// TwinCAT 3 PLC project OSCAT
// Title: OSCAT
// Company: RWTH Aachen University - E.ON Energy Research Center
// ProjectVersion: 1.1.3
// Description: This library is based on the OSCAT library (http://www.oscat.de/)
// ProgramVersion: 3.1.4022.1
// libraries:
//   Tc2_Standard, * (Beckhoff Automation GmbH)
// project tree:
//   oscat_basic/Data types/ CALENDAR.TcDUT (not stored), COMPLEX.TcDUT (not stored), CONSTANTS_LANGUAGE.TcDUT (not stored), CONSTANTS_LOCATION.TcDUT (not stored), CONSTANTS_MATH.TcDUT (not stored), CONSTANTS_PHYS.TcDUT (not stored), CONSTANTS_SETUP.TcDUT (not stored), ESR_DATA.TcDUT (not stored), CONTROL_MODE.TcDUT (not stored), FRACTION.TcDUT (not stored), HOLIDAY_DATA.TcDUT (not stored), REAL2.TcDUT (not stored), SDT.TcDUT (not stored), CONTROL_PARAMETERS.TcDUT (not stored), IO_TERMINAL_PARAMETERS.TcDUT (not stored), TIMER_EVENT.TcDUT (not stored), VECTOR_3.TcDUT (not stored)
//   oscat_basic/Global Variables/ Constants_2.TcGVL (not stored), Globale_Variablen_2.TcGVL (not stored)
//   oscat_basic/POUs/Buffer Management/ BUFFER_COMP.TcPOU (not stored), BUFFER_SEARCH.TcPOU (not stored), BUFFER_TO_STRING.TcPOU (not stored), _BUFFER_INSERT.TcPOU (not stored), _BUFFER_UPPERCASE.TcPOU (not stored), _STRING_TO_BUFFER.TcPOU (not stored)
//   oscat_basic/POUs/Engineering/automation/ DRIVER_1.TcPOU (not stored), DRIVER_4.TcPOU (not stored), DRIVER_4C.TcPOU (not stored), FLOW_CONTROL.TcPOU (not stored), FT_Profile.TcPOU (not stored), INC_DEC.TcPOU (not stored), INTERLOCK.TcPOU (not stored), INTERLOCK_4.TcPOU (not stored), MANUAL.TcPOU (not stored), MANUAL_1.TcPOU (not stored), MANUAL_2.TcPOU (not stored), MANUAL_4.TcPOU (not stored), PARSET.TcPOU (not stored), PARSET2.TcPOU (not stored), SIGNAL.TcPOU (not stored), SIGNAL_4.TcPOU (not stored), SRAMP.TcPOU (not stored), TUNE.TcPOU (not stored), TUNE2.TcPOU (not stored)
//   oscat_basic/POUs/Engineering/Control/ BAND_B.TcPOU (not stored), CONTROL_SET1.TcPOU (not stored), CONTROL_SET2.TcPOU (not stored), CTRL_IN.TcPOU (not stored), CTRL_OUT.TcPOU (not stored), CTRL_PI.TcPOU (not stored), CTRL_PID.TcPOU (not stored), CTRL_PWM.TcPOU (not stored), DEAD_BAND.TcPOU (not stored), DEAD_BAND_A.TcPOU (not stored), DEAD_ZONE.TcPOU (not stored), DEAD_ZONE2.TcPOU (not stored), VOLTAGE_CONTROL.TcPOU (not stored), FB_CONTROL.TcPOU (not stored), FB_Integrate.TcPOU (not stored), FB_PID.TcPOU (not stored), FT_DERIV.TcPOU (not stored), FT_IMP.TcPOU (not stored), FT_INT.TcPOU (not stored), FT_INT2.TcPOU (not stored), FT_PD.TcPOU (not stored), FT_PDT1.TcPOU (not stored), FT_PI.TcPOU (not stored), FT_PID.TcPOU (not stored), FT_PIDW.TcPOU (not stored), FT_PIDWL.TcPOU (not stored), FT_PIW.TcPOU (not stored), FT_PIWL.TcPOU (not stored), FT_PT1.TcPOU (not stored), FT_PT2.TcPOU (not stored), FT_TN16.TcPOU (not stored), FT_TN64.TcPOU (not stored), FT_TN8.TcPOU (not stored), HYST.TcPOU (not stored), HYST_1.TcPOU (not stored), HYST_2.TcPOU (not stored), HYST_3.TcPOU (not stored), INTEGRATE.TcPOU (not stored)
//   oscat_basic/POUs/Engineering/Conversion/ ASTRO.TcPOU (not stored), BFT_TO_MS.TcPOU (not stored), C_TO_F.TcPOU (not stored), C_TO_K.TcPOU (not stored), DEG_TO_DIR.TcPOU (not stored), DIR_TO_DEG.TcPOU (not stored), ENERGY.TcPOU (not stored), F_TO_C.TcPOU (not stored), F_TO_OM.TcPOU (not stored), F_TO_PT.TcPOU (not stored), GEO_TO_DEG.TcPOU (not stored), KMH_TO_MS.TcPOU (not stored), K_TO_C.TcPOU (not stored), LENGTH.TcPOU (not stored), MS_TO_BFT.TcPOU (not stored), MS_TO_KMH.TcPOU (not stored), OM_TO_F.TcPOU (not stored), PRESSURE.TcPOU (not stored), PT_TO_F.TcPOU (not stored), SPEED.TcPOU (not stored), TEMPERATURE.TcPOU (not stored)
//   oscat_basic/POUs/Engineering/measurements/ ALARM_2.TcPOU (not stored), BAR_GRAPH.TcPOU (not stored), CALIBRATE.TcPOU (not stored), CYCLE_TIME.TcPOU (not stored), DT_SIMU.TcPOU (not stored), FLOW_METER.TcPOU (not stored), METER.TcPOU (not stored), METER_STAT.TcPOU (not stored), M_D.TcPOU (not stored), M_T.TcPOU (not stored), M_TX.TcPOU (not stored), ONTIME.TcPOU (not stored), TC_MS.TcPOU (not stored), TC_S.TcPOU (not stored), TC_US.TcPOU (not stored), T_PLC_MS.TcPOU (not stored), T_PLC_US.TcPOU (not stored)
//   oscat_basic/POUs/Engineering/sensor/ MULTI_IN.TcPOU (not stored), RES_NI.TcPOU (not stored), RES_NTC.TcPOU (not stored), RES_PT.TcPOU (not stored), RES_SI.TcPOU (not stored), SENSOR_INT.TcPOU (not stored), TEMP_NI.TcPOU (not stored), TEMP_NTC.TcPOU (not stored), TEMP_PT.TcPOU (not stored), TEMP_SI.TcPOU (not stored)
//   oscat_basic/POUs/Engineering/signal generators/ GEN_PULSE.TcPOU (not stored), GEN_PW2.TcPOU (not stored), GEN_RDM.TcPOU (not stored), GEN_RDT.TcPOU (not stored), GEN_RMP.TcPOU (not stored), GEN_SIN.TcPOU (not stored), GEN_SQR.TcPOU (not stored), PWM_DC.TcPOU (not stored), PWM_PW.TcPOU (not stored), RMP_B.TcPOU (not stored), RMP_SOFT.TcPOU (not stored), RMP_W.TcPOU (not stored), _RMP_B.TcPOU (not stored), _RMP_NEXT.TcPOU (not stored), _RMP_W.TcPOU (not stored)
//   oscat_basic/POUs/Engineering/signal processing/ AIN.TcPOU (not stored), AIN1.TcPOU (not stored), AOUT.TcPOU (not stored), AOUT1.TcPOU (not stored), BYTE_TO_RANGE.TcPOU (not stored), DELAY.TcPOU (not stored), DELAY_200.TcPOU (not stored), DELAY_4.TcPOU (not stored), FADE.TcPOU (not stored), FB_InLinear.TcPOU (not stored), FB_InOnOff.TcPOU (not stored), FB_OutLinear.TcPOU (not stored), FB_OutOnOff.TcPOU (not stored), FILTER_DW.TcPOU (not stored), FILTER_I.TcPOU (not stored), FILTER_MAV_DW.TcPOU, FILTER_MAV_W.TcPOU (not stored), FILTER_W.TcPOU (not stored), FILTER_WAV.TcPOU (not stored), MIX.TcPOU (not stored), MUX_R2.TcPOU (not stored), MUX_R4.TcPOU (not stored), OFFSET.TcPOU (not stored), OFFSET2.TcPOU (not stored), OVERRIDE.TcPOU (not stored), RANGE_TO_BYTE.TcPOU (not stored), RANGE_TO_WORD.TcPOU (not stored), SCALE.TcPOU (not stored), SCALE_B.TcPOU (not stored), SCALE_B2.TcPOU (not stored), SCALE_B4.TcPOU (not stored), SCALE_B8.TcPOU (not stored), SCALE_D.TcPOU (not stored), SCALE_R.TcPOU (not stored), SCALE_X2.TcPOU (not stored), SCALE_X4.TcPOU (not stored), SCALE_X8.TcPOU (not stored), SEL2_OF_3.TcPOU (not stored), SEL2_OF_3B.TcPOU (not stored), SH.TcPOU (not stored), SH_1.TcPOU (not stored), SH_2.TcPOU (not stored), SH_T.TcPOU (not stored), STAIR.TcPOU (not stored), STAIR2.TcPOU (not stored), TREND.TcPOU (not stored), TREND_DW.TcPOU (not stored), WORD_TO_RANGE.TcPOU (not stored)
//   oscat_basic/POUs/List Processing/ LIST_ADD.TcPOU (not stored), LIST_CLEAN.TcPOU (not stored), LIST_GET.TcPOU (not stored), LIST_INSERT.TcPOU (not stored), LIST_LEN.TcPOU (not stored), LIST_NEXT.TcPOU (not stored), LIST_RETRIEVE.TcPOU (not stored), LIST_RETRIEVE_LAST.TcPOU (not stored)
//   oscat_basic/POUs/Logic/FF edge triggered/ COUNT_BR.TcPOU (not stored), COUNT_DR.TcPOU (not stored), FF_D2E.TcPOU (not stored), FF_D4E.TcPOU (not stored), FF_DRE.TcPOU (not stored), FF_JKE.TcPOU (not stored), FF_RSE.TcPOU (not stored), SELECT_8.TcPOU (not stored), SHR_4E.TcPOU (not stored), SHR_4UDE.TcPOU (not stored), SHR_8PLE.TcPOU (not stored), SHR_8UDE.TcPOU (not stored), TOGGLE.TcPOU (not stored)
//   oscat_basic/POUs/Logic/FF pulse triggered/ LTCH.TcPOU (not stored), LTCH_4.TcPOU (not stored), STORE_8.TcPOU (not stored)
//   oscat_basic/POUs/Logic/gate logic/ BCDC_TO_INT.TcPOU (not stored), BIT_COUNT.TcPOU (not stored), BIT_LOAD_B.TcPOU (not stored), BIT_LOAD_B2.TcPOU (not stored), BIT_LOAD_DW.TcPOU (not stored), BIT_LOAD_DW2.TcPOU (not stored), BIT_LOAD_W.TcPOU (not stored), BIT_LOAD_W2.TcPOU (not stored), BIT_OF_DWORD.TcPOU (not stored), BIT_TOGGLE_B.TcPOU (not stored), BIT_TOGGLE_DW.TcPOU (not stored), BIT_TOGGLE_W.TcPOU (not stored), BYTE_OF_BIT.TcPOU (not stored), BYTE_OF_DWORD.TcPOU (not stored), BYTE_TO_BITS.TcPOU (not stored), BYTE_TO_GRAY.TcPOU (not stored), CHECK_PARITY.TcPOU (not stored), CHK_REAL.TcPOU (not stored), DEC_2.TcPOU (not stored), DEC_4.TcPOU (not stored), DEC_8.TcPOU (not stored), DWORD_OF_BYTE.TcPOU (not stored), DWORD_OF_WORD.TcPOU (not stored), DW_TO_REAL.TcPOU (not stored), GRAY_TO_BYTE.TcPOU (not stored), INT_TO_BCDC.TcPOU (not stored), MUX_2.TcPOU (not stored), MUX_4.TcPOU (not stored), PARITY.TcPOU (not stored), REAL_TO_DW.TcPOU (not stored), REFLECT.TcPOU (not stored), REVERSE.TcPOU (not stored), SHL1.TcPOU (not stored), SHR1.TcPOU (not stored), SWAP_BYTE.TcPOU (not stored), SWAP_BYTE2.TcPOU (not stored), WORD_OF_BYTE.TcPOU (not stored), WORD_OF_DWORD.TcPOU (not stored)
//   oscat_basic/POUs/Logic/generators/ A_TRIG.TcPOU (not stored), B_TRIG.TcPOU (not stored), CLICK_CNT.TcPOU (not stored), CLICK_DEC.TcPOU (not stored), CLK_DIV.TcPOU (not stored), CLK_N.TcPOU (not stored), CLK_PRG.TcPOU (not stored), CLK_PULSE.TcPOU (not stored), CYCLE_4.TcPOU (not stored), D_TRIG.TcPOU (not stored), GEN_BIT.TcPOU (not stored), GEN_SQ.TcPOU (not stored), SCHEDULER.TcPOU (not stored), SCHEDULER_2.TcPOU (not stored), SEQUENCE_4.TcPOU (not stored), SEQUENCE_64.TcPOU (not stored), SEQUENCE_8.TcPOU (not stored), TMAX.TcPOU (not stored), TMIN.TcPOU (not stored), TOF_1.TcPOU (not stored), TONOF.TcPOU (not stored), TP_1.TcPOU (not stored), TP_1D.TcPOU (not stored), TP_X.TcPOU (not stored)
//   oscat_basic/POUs/Logic/memory/ FIFO_16.TcPOU (not stored), FIFO_32.TcPOU (not stored), STACK_16.TcPOU (not stored), STACK_32.TcPOU (not stored)
//   oscat_basic/POUs/Logic/Others/ CRC_GEN.TcPOU (not stored), MATRIX.TcPOU (not stored), PIN_CODE.TcPOU (not stored)
//   oscat_basic/POUs/Mathematical/ ACOSH.TcPOU (not stored), ACOTH.TcPOU (not stored), AGDF.TcPOU (not stored), ASINH.TcPOU (not stored), ATAN2.TcPOU (not stored), ATANH.TcPOU (not stored), BETA.TcPOU (not stored), BINOM.TcPOU (not stored), CAUCHY.TcPOU (not stored), CAUCHYCD.TcPOU (not stored), CEIL.TcPOU (not stored), CEIL2.TcPOU (not stored), CMP.TcPOU (not stored), COSH.TcPOU (not stored), COTH.TcPOU (not stored), DEC1.TcPOU (not stored), DEG.TcPOU (not stored), DIFFER.TcPOU (not stored), D_TRUNC.TcPOU (not stored), ERF.TcPOU (not stored), ERFC.TcPOU (not stored), EVEN.TcPOU (not stored), EXP10.TcPOU (not stored), EXPN.TcPOU (not stored), FACT.TcPOU (not stored), FIB.TcPOU (not stored), FLOOR.TcPOU (not stored), FLOOR2.TcPOU (not stored), FRACT.TcPOU (not stored), GAMMA.TcPOU (not stored), GAUSS.TcPOU (not stored), GAUSSCD.TcPOU (not stored), GCD.TcPOU (not stored), GDF.TcPOU (not stored), GOLD.TcPOU (not stored), HYPOT.TcPOU (not stored), INC.TcPOU (not stored), INC1.TcPOU (not stored), INC2.TcPOU (not stored), INV.TcPOU (not stored), LAMBERT_W.TcPOU (not stored), LANGEVIN.TcPOU (not stored), MAX3.TcPOU (not stored), MID3.TcPOU (not stored), MIN3.TcPOU (not stored), MODR.TcPOU (not stored), MUL_ADD.TcPOU (not stored), NEGX.TcPOU (not stored), RAD.TcPOU (not stored), RDM.TcPOU (not stored), RDM2.TcPOU (not stored), RDMDW.TcPOU (not stored), REAL_TO_FRAC.TcPOU (not stored), RND.TcPOU (not stored), ROUND.TcPOU (not stored), SGN.TcPOU (not stored), SIGMOID.TcPOU (not stored), SIGN_I.TcPOU (not stored), SIGN_R.TcPOU (not stored), SINC.TcPOU (not stored), SINH.TcPOU (not stored), SQRTN.TcPOU (not stored), TANC.TcPOU (not stored), TANH.TcPOU (not stored), WINDOW.TcPOU (not stored), WINDOW2.TcPOU (not stored)
//   oscat_basic/POUs/Mathematical/Array/ ARRAY_AVG.TcPOU (not stored), ARRAY_GAV.TcPOU (not stored), ARRAY_HAV.TcPOU (not stored), ARRAY_MAX.TcPOU (not stored), ARRAY_MIN.TcPOU (not stored), ARRAY_SDV.TcPOU (not stored), ARRAY_SPR.TcPOU (not stored), ARRAY_SUM.TcPOU (not stored), ARRAY_TREND.TcPOU (not stored), ARRAY_VAR.TcPOU (not stored), IS_SORTED.TcPOU (not stored), _ARRAY_ABS.TcPOU (not stored), _ARRAY_ADD.TcPOU (not stored), _ARRAY_INIT.TcPOU (not stored), _ARRAY_MEDIAN.TcPOU (not stored), _ARRAY_MUL.TcPOU (not stored), _ARRAY_SHUFFLE.TcPOU (not stored), _ARRAY_SORT.TcPOU (not stored)
//   oscat_basic/POUs/Mathematical/Complex/ CABS.TcPOU (not stored), CACOS.TcPOU (not stored), CACOSH.TcPOU (not stored), CADD.TcPOU (not stored), CARG.TcPOU (not stored), CASIN.TcPOU (not stored), CASINH.TcPOU (not stored), CATAN.TcPOU (not stored), CATANH.TcPOU (not stored), CCON.TcPOU (not stored), CCOS.TcPOU (not stored), CCOSH.TcPOU (not stored), CDIV.TcPOU (not stored), CEXP.TcPOU (not stored), CINV.TcPOU (not stored), CLOG.TcPOU (not stored), CMUL.TcPOU (not stored), CPOL.TcPOU (not stored), CPOW.TcPOU (not stored), CSET.TcPOU (not stored), CSIN.TcPOU (not stored), CSINH.TcPOU (not stored), CSQRT.TcPOU (not stored), CSUB.TcPOU (not stored), CTAN.TcPOU (not stored), CTANH.TcPOU (not stored)
//   oscat_basic/POUs/Mathematical/Double Precision/ R2_ABS.TcPOU (not stored), R2_ADD.TcPOU (not stored), R2_ADD2.TcPOU (not stored), R2_MUL.TcPOU (not stored), R2_SET.TcPOU (not stored)
//   oscat_basic/POUs/Mathematical/functions/ FRMP_B.TcPOU (not stored), FT_AVG.TcPOU (not stored), FT_AVG_200.TcPOU (not stored), FT_MIN_MAX.TcPOU (not stored), FT_RMP.TcPOU (not stored), F_LIN.TcPOU (not stored), F_LIN2.TcPOU (not stored), F_POLY.TcPOU (not stored), F_POWER.TcPOU (not stored), F_QUAD.TcPOU (not stored), LINEAR_INT.TcPOU (not stored), POLYNOM_INT.TcPOU (not stored)
//   oscat_basic/POUs/Mathematical/Geometry/ CIRCLE_A.TcPOU (not stored), CIRCLE_C.TcPOU (not stored), CIRCLE_SEG.TcPOU (not stored), CONE_V.TcPOU (not stored), ELLIPSE_A.TcPOU (not stored), ELLIPSE_C.TcPOU (not stored), SPHERE_V.TcPOU (not stored), TRIANGLE_A.TcPOU (not stored)
//   oscat_basic/POUs/Mathematical/Vektormathematik/ V3_ABS.TcPOU (not stored), V3_ADD.TcPOU (not stored), V3_ANG.TcPOU (not stored), V3_DPRO.TcPOU (not stored), V3_NORM.TcPOU (not stored), V3_NUL.TcPOU (not stored), V3_PAR.TcPOU (not stored), V3_REV.TcPOU (not stored), V3_SMUL.TcPOU (not stored), V3_SUB.TcPOU (not stored), V3_XANG.TcPOU (not stored), V3_XPRO.TcPOU (not stored), V3_YANG.TcPOU (not stored), V3_ZANG.TcPOU (not stored)
//   oscat_basic/POUs/Other/ ESR_COLLECT.TcPOU (not stored), ESR_MON_B8.TcPOU (not stored), ESR_MON_R4.TcPOU (not stored), ESR_MON_X8.TcPOU (not stored), OSCAT_VERSION.TcPOU (not stored), STATUS_TO_ESR.TcPOU (not stored)
//   oscat_basic/POUs/String/ BIN_TO_BYTE.TcPOU (not stored), BIN_TO_DWORD.TcPOU (not stored), BYTE_TO_STRB.TcPOU (not stored), BYTE_TO_STRH.TcPOU (not stored), CAPITALIZE.TcPOU (not stored), CHARCODE.TcPOU (not stored), CHARNAME.TcPOU (not stored), CHR_TO_STRING.TcPOU (not stored), CLEAN.TcPOU (not stored), CODE.TcPOU (not stored), COUNT_CHAR.TcPOU (not stored), COUNT_SUBSTRING.TcPOU (not stored), DEC_TO_BYTE.TcPOU (not stored), DEC_TO_DWORD.TcPOU (not stored), DEC_TO_INT.TcPOU (not stored), DEL_CHARS.TcPOU (not stored), DT_TO_STRF.TcPOU (not stored), DWORD_TO_STRB.TcPOU (not stored), DWORD_TO_STRF.TcPOU (not stored), DWORD_TO_STRH.TcPOU (not stored), EXEC.TcPOU (not stored), FILL.TcPOU (not stored), FINDB.TcPOU (not stored), FINDB_NONUM.TcPOU (not stored), FINDB_NUM.TcPOU (not stored), FINDP.TcPOU (not stored), FIND_CHAR.TcPOU (not stored), FIND_CTRL.TcPOU (not stored), FIND_NONUM.TcPOU (not stored), FIND_NUM.TcPOU (not stored), FIX.TcPOU (not stored), FLOAT_TO_REAL.TcPOU (not stored), FSTRING_TO_BYTE.TcPOU (not stored), FSTRING_TO_DT.TcPOU (not stored), FSTRING_TO_DWORD.TcPOU (not stored), FSTRING_TO_MONTH.TcPOU (not stored), FSTRING_TO_WEEK.TcPOU (not stored), FSTRING_TO_WEEKDAY.TcPOU (not stored), HEX_TO_BYTE.TcPOU (not stored), HEX_TO_DWORD.TcPOU (not stored), ISC_ALPHA.TcPOU (not stored), ISC_CTRL.TcPOU (not stored), ISC_HEX.TcPOU (not stored), ISC_LOWER.TcPOU (not stored), ISC_NUM.TcPOU (not stored), ISC_UPPER.TcPOU (not stored), IS_ALNUM.TcPOU (not stored), IS_ALPHA.TcPOU (not stored), IS_CC.TcPOU (not stored), IS_CTRL.TcPOU (not stored), IS_HEX.TcPOU (not stored), IS_LOWER.TcPOU (not stored), IS_NCC.TcPOU (not stored), IS_NUM.TcPOU (not stored), IS_UPPER.TcPOU (not stored), LOWERCASE.TcPOU (not stored), MESSAGE_4R.TcPOU (not stored), MESSAGE_8.TcPOU (not stored), MIRROR.TcPOU (not stored), MONTH_TO_STRING.TcPOU (not stored), OCT_TO_BYTE.TcPOU (not stored), OCT_TO_DWORD.TcPOU (not stored), REAL_TO_STRF.TcPOU (not stored), REPLACE_ALL.TcPOU (not stored), REPLACE_CHARS.TcPOU (not stored), REPLACE_UML.TcPOU (not stored), TICKER.TcPOU (not stored), TO_LOWER.TcPOU (not stored), TO_UML.TcPOU (not stored), TO_UPPER.TcPOU (not stored), TRIM.TcPOU (not stored), TRIM1.TcPOU (not stored), TRIME.TcPOU (not stored), UPPERCASE.TcPOU (not stored), WEEKDAY_TO_STRING.TcPOU (not stored)
//   oscat_basic/POUs/Time&Date/ CALENDAR_CALC.TcPOU (not stored), DATE_ADD.TcPOU (not stored), DAYS_DELTA.TcPOU (not stored), DAYS_IN_MONTH.TcPOU (not stored), DAYS_IN_YEAR.TcPOU (not stored), DAY_OF_DATE.TcPOU (not stored), DAY_OF_MONTH.TcPOU (not stored), DAY_OF_WEEK.TcPOU (not stored), DAY_OF_YEAR.TcPOU (not stored), DAY_TO_TIME.TcPOU (not stored), DCF77.TcPOU (not stored), DST.TcPOU (not stored), DT2_TO_SDT.TcPOU (not stored), DT_TO_SDT.TcPOU (not stored), EASTER.TcPOU (not stored), EVENTS.TcPOU (not stored), HOLIDAY.TcPOU (not stored), HOUR.TcPOU (not stored), HOUR_OF_DT.TcPOU (not stored), HOUR_TO_TIME.TcPOU (not stored), HOUR_TO_TOD.TcPOU (not stored), JD2000.TcPOU (not stored), LEAP_DAY.TcPOU (not stored), LEAP_OF_DATE.TcPOU (not stored), LEAP_YEAR.TcPOU (not stored), LTIME_TO_UTC.TcPOU (not stored), MINUTE.TcPOU (not stored), MINUTE_OF_DT.TcPOU (not stored), MINUTE_TO_TIME.TcPOU (not stored), MONTH_BEGIN.TcPOU (not stored), MONTH_END.TcPOU (not stored), MONTH_OF_DATE.TcPOU (not stored), MULTIME.TcPOU (not stored), PERIOD.TcPOU (not stored), PERIOD2.TcPOU (not stored), REFRACTION.TcPOU (not stored), RTC_2.TcPOU (not stored), RTC_MS.TcPOU (not stored), SDT_TO_DATE.TcPOU (not stored), SDT_TO_DT.TcPOU (not stored), SDT_TO_TOD.TcPOU (not stored), SECOND.TcPOU (not stored), SECOND_OF_DT.TcPOU (not stored), SECOND_TO_TIME.TcPOU (not stored), SET_DATE.TcPOU (not stored), SET_DT.TcPOU (not stored), SET_TOD.TcPOU (not stored), SUN_MIDDAY.TcPOU (not stored), SUN_POS.TcPOU (not stored), SUN_TIME.TcPOU (not stored), TIMECHECK.TcPOU (not stored), TON_P.TcPOU (not stored), UTC_TO_LTIME.TcPOU (not stored), WORK_WEEK.TcPOU (not stored), YEAR_BEGIN.TcPOU (not stored), YEAR_END.TcPOU (not stored), YEAR_OF_DATE.TcPOU (not stored)
//   oscat_building/Global Variables/ Constants.TcGVL (not stored), Globale_Variablen.TcGVL (not stored), Setup_Data.TcGVL (not stored)
//   oscat_building/POUs/actuators/ ACTUATOR_2P.TcPOU (not stored), ACTUATOR_3P.TcPOU (not stored), ACTUATOR_A.TcPOU (not stored), ACTUATOR_COIL.TcPOU (not stored), ACTUATOR_PUMP.TcPOU (not stored), ACTUATOR_UD.TcPOU (not stored), AUTORUN.TcPOU (not stored)
//   oscat_building/POUs/electrical/ CLICK.TcPOU (not stored), CLICK_MODE.TcPOU (not stored), DEBOUNCE.TcPOU (not stored), DIMM_2.TcPOU (not stored), DIMM_I.TcPOU (not stored), F_LAMP.TcPOU (not stored), PULSE_LENGTH.TcPOU (not stored), PULSE_T.TcPOU (not stored), SWITCH_I.TcPOU (not stored), SWITCH_X.TcPOU (not stored), SW_RECONFIG.TcPOU (not stored), TIMER_1.TcPOU (not stored), TIMER_2.TcPOU (not stored), TIMER_EVENT_DECODE.TcPOU (not stored), TIMER_EXT.TcPOU (not stored), TIMER_P4.TcPOU (not stored)
//   oscat_building/POUs/HLK/ AIR_DENSITY.TcPOU (not stored), AIR_ENTHALPY.TcPOU (not stored), BOILER.TcPOU (not stored), BURNER.TcPOU (not stored), DEW_CON.TcPOU (not stored), DEW_RH.TcPOU (not stored), DEW_TEMP.TcPOU (not stored), HEAT_INDEX.TcPOU (not stored), HEAT_METER.TcPOU (not stored), HEAT_TEMP.TcPOU (not stored), LEGIONELLA.TcPOU (not stored), SDD.TcPOU (not stored), SDD_NH3.TcPOU (not stored), SDT_NH3.TcPOU (not stored), TANK_LEVEL.TcPOU (not stored), TANK_VOL1.TcPOU (not stored), TANK_VOL2.TcPOU (not stored), TEMP_EXT.TcPOU (not stored), T_AVG24.TcPOU (not stored), WATER_CP.TcPOU (not stored), WATER_DENSITY.TcPOU (not stored), WATER_ENTHALPY.TcPOU (not stored), WCT.TcPOU (not stored)
//   oscat_building/POUs/Jalousie/ BLIND_ACTUATOR.TcPOU (not stored), BLIND_CONTROL.TcPOU (not stored), BLIND_CONTROL_S.TcPOU (not stored), BLIND_INPUT.TcPOU (not stored), BLIND_NIGHT.TcPOU (not stored), BLIND_SCENE.TcPOU (not stored), BLIND_SECURITY.TcPOU (not stored), BLIND_SET.TcPOU (not stored), BLIND_SHADE.TcPOU (not stored), BLIND_SHADE_S.TcPOU (not stored)
//   oscat_building/POUs/Other/ BUILDING_VERSION.TcPOU (not stored)
//   oscat_network/Data types/DATA_LOG/ DLOG_DATA.TcDUT (not stored), LOG_CONTROL.TcDUT (not stored), MYSQL_COM.TcDUT (not stored), PRINTF_DATA.TcDUT (not stored), UNI_CIRCULAR_BUFFER_DATA.TcDUT (not stored), us_LOG_VIEWPORT.TcDUT (not stored)
//   oscat_network/Data types/FILE_SERVER/ FILE_PATH_DATA.TcDUT (not stored), FILE_SERVER_DATA.TcDUT (not stored)
//   oscat_network/Data types/NETWORK/ IP2GEO_DATA.TcDUT (not stored), IP_C.TcDUT (not stored), IP_FIFO_DATA.TcDUT (not stored), NETWORK_BUFFER.TcDUT (not stored), NETWORK_BUFFER_SHORT.TcDUT (not stored), NW_BUF_LONG.TcDUT (not stored), NW_BUF_SHORT.TcDUT (not stored), URL.TcDUT (not stored), VMAP_DATA.TcDUT (not stored), XML_CONTROL.TcDUT (not stored)
//   oscat_network/Data types/NET_VAR/ NET_VAR_DATA.TcDUT (not stored)
//   oscat_network/Data types/TELNET_VISION/ us_TN_INPUT_CONTROL.TcDUT (not stored), us_TN_INPUT_CONTROL_DATA.TcDUT (not stored), us_TN_MENU.TcDUT (not stored), us_TN_MENU_POPUP.TcDUT (not stored), us_TN_SCREEN.TcDUT (not stored)
//   oscat_network/Data types/WEATHER/ WORLD_WEATHER_CUR.TcDUT (not stored), WORLD_WEATHER_DATA.TcDUT (not stored), WORLD_WEATHER_DAY.TcDUT (not stored), YAHOO_WEATHER_DATA.TcDUT (not stored)
//   oscat_network/Global Variables/ Constants_1.TcGVL (not stored), Globale_Variablen_1.TcGVL (not stored)
//   oscat_network/POUs/CO_NVERT/ BASE64_DECODE_STREAM_1.TcPOU (not stored), BASE64_DECODE_STR_1.TcPOU (not stored), BASE64_ENCODE_STREAM_1.TcPOU (not stored), BASE64_ENCODE_STR_1.TcPOU (not stored), HTML_DECODE_1.TcPOU (not stored), HTML_ENCODE_1.TcPOU (not stored), IP4_CHECK_1.TcPOU (not stored), IP4_DECODE_1.TcPOU (not stored), IP4_TO_STRING_1.TcPOU (not stored), IS_IP4_1.TcPOU (not stored), IS_URLCHR_1.TcPOU (not stored), MD5_AUX_1.TcPOU (not stored), MD5_CRAM_AUTH_1.TcPOU (not stored), MD5_STREAM_1.TcPOU (not stored), MD5_STR_1.TcPOU (not stored), MD5_TO_STRH_1.TcPOU (not stored), RC4_CRYPT_STREAM_1.TcPOU (not stored), SHA1_STREAM_1.TcPOU (not stored), SHA1_STR_1.TcPOU (not stored), SHA1_TO_STRH_1.TcPOU (not stored), STRING_TO_URL_1.TcPOU (not stored), URL_DECODE_1.TcPOU (not stored), URL_ENCODE_1.TcPOU (not stored), URL_TO_STRING_1.TcPOU (not stored)
//   oscat_network/POUs/DATA_LOG/ DLOG_BOOL_1.TcPOU (not stored), DLOG_DINT_1.TcPOU (not stored), DLOG_DT_1.TcPOU (not stored), DLOG_FILE_TO_FTP_1.TcPOU (not stored), DLOG_FILE_TO_SMTP_1.TcPOU (not stored), DLOG_REAL_1.TcPOU (not stored), DLOG_STORE_FILE_CSV_1.TcPOU (not stored), DLOG_STORE_FILE_HTML_1.TcPOU (not stored), DLOG_STORE_FILE_XML_1.TcPOU (not stored), DLOG_STORE_RRD_1.TcPOU (not stored), DLOG_STRING_1.TcPOU (not stored), UNI_CIRCULAR_BUFFER_1.TcPOU (not stored)
//   oscat_network/POUs/DEMO/ BASE64_DEMO_1.TcPOU (not stored), CSV_PARSER_BUF_DEMO_1.TcPOU (not stored), CSV_PARSER_FILE_DEMO_1.TcPOU (not stored), DLOG_FILE_CSV_DEMO_1.TcPOU (not stored), DLOG_FILE_CSV_FTP_DEMO_1.TcPOU (not stored), DLOG_FILE_CSV_SMTP_DEMO_1.TcPOU (not stored), DLOG_FILE_HTML_DEMO_1.TcPOU (not stored), DLOG_FILE_XML_DEMO_1.TcPOU (not stored), DLOG_RRD_DEMO_1.TcPOU (not stored), DNS_DYN_DEMO_1.TcPOU (not stored), DNS_REV_DEMO_1.TcPOU (not stored), DNS_SNTP_SYSLOG_DEMO_1.TcPOU (not stored), FILE_BLOCK_DEMO_1.TcPOU (not stored), FTP_CLIENT_DEMO_1.TcPOU (not stored), GET_WAN_IP_DEMO_1.TcPOU (not stored), HTTP_DEMO_1.TcPOU (not stored), INI_PARSER_BUF_DEMO_1.TcPOU (not stored), INI_PARSER_FILE_DEMO_1.TcPOU (not stored), IP2GEO_DEMO_1.TcPOU (not stored), IRTRANS_DEMO_1.TcPOU (not stored), MB_CLIENT_DEMO_1.TcPOU (not stored), MB_SERVER_DEMO_1.TcPOU (not stored), MD5_CRAM_AUTH_DEMO_1.TcPOU (not stored), NET_VAR_MASTER_DEMO_1.TcPOU (not stored), NET_VAR_SLAVE_DEMO_1.TcPOU (not stored), RC4_CRYPT_DEMO_1.TcPOU (not stored), SHA1_MD5_DEMO_1.TcPOU (not stored), SMTP_CLIENT_DEMO_1.TcPOU (not stored), SPIDER_DEMO_1.TcPOU (not stored), TELNET_LOG_DEMO_1.TcPOU (not stored), TELNET_PRINT_DEMO_1.TcPOU (not stored), TN_VISION_DEMO_1_1.TcPOU (not stored), TN_VISION_DEMO_2_1.TcPOU (not stored), WORLD_WEATHER_DEMO_1.TcPOU (not stored), YAHOO_WEATHER_DEMO_1.TcPOU (not stored)
//   oscat_network/POUs/DRIVER/ IRTRANS_DECODE_1.TcPOU (not stored), IRTRANS_RCV_1_1.TcPOU (not stored), IRTRANS_RCV_4_1.TcPOU (not stored), IRTRANS_RCV_8_1.TcPOU (not stored), IRTRANS_SERVER_1.TcPOU (not stored), IRTRANS_SND_1_1.TcPOU (not stored), IRTRANS_SND_4_1.TcPOU (not stored), IRTRANS_SND_8_1.TcPOU (not stored)
//   oscat_network/POUs/FILE/ CSV_PARSER_BUF_1.TcPOU (not stored), CSV_PARSER_FILE_1.TcPOU (not stored), FILE_BLOCK_1.TcPOU (not stored), FILE_PATH_SPLIT_1.TcPOU (not stored), INI_PARSER_BUF_1.TcPOU (not stored), INI_PARSER_FILE_1.TcPOU (not stored)
//   oscat_network/POUs/HARDWARE/ FILE_SERVER_1.TcPOU (not stored), IP_CONTROL2_1.TcPOU (not stored), IP_CONTROL_1.TcPOU (not stored), IP_CONTROL_RESET_1.TcPOU (not stored)
//   oscat_network/POUs/NETWORK/ DNS_CLIENT.TcPOU (not stored), DNS_DYN.TcPOU (not stored), DNS_REV_CLIENT.TcPOU (not stored), FTP_CLIENT.TcPOU (not stored), GET_WAN_IP.TcPOU (not stored), HTTP_GET.TcPOU (not stored), IP2GEO.TcPOU (not stored), IP_FIFO.TcPOU (not stored), LOG_MSG.TcPOU (not stored), LOG_VIEWPORT.TcPOU (not stored), MB_CLIENT.TcPOU (not stored), MB_SERVER.TcPOU (not stored), MB_VMAP.TcPOU (not stored), PRINT_SF.TcPOU (not stored), READ_HTTP.TcPOU (not stored), SMTP_CLIENT.TcPOU (not stored), SNTP_CLIENT.TcPOU (not stored), SNTP_SERVER.TcPOU (not stored), SPIDER_ACCESS.TcPOU (not stored), SYS_LOG.TcPOU (not stored), TELNET_LOG.TcPOU (not stored), TELNET_PRINT.TcPOU (not stored), XML_READER.TcPOU (not stored)
//   oscat_network/POUs/NET_VAR/ NET_VAR_BOOL8.TcPOU (not stored), NET_VAR_BUFFER.TcPOU (not stored), NET_VAR_CONTROL.TcPOU (not stored), NET_VAR_DWORD8.TcPOU (not stored), NET_VAR_REAL8.TcPOU (not stored), NET_VAR_STRING.TcPOU (not stored), NET_VAR_X8.TcPOU (not stored)
//   oscat_network/POUs/OTHER/ ELEMENT_COUNT.TcPOU (not stored), ELEMENT_GET.TcPOU (not stored), NETWORK_VERSION.TcPOU (not stored)
//   oscat_network/POUs/TELNET_VISION/ TN_FRAMEWORK.TcPOU (not stored), TN_INPUT_CONTROL.TcPOU (not stored), TN_INPUT_EDIT_LINE.TcPOU (not stored), TN_INPUT_MENU_BAR.TcPOU (not stored), TN_INPUT_MENU_POPUP.TcPOU (not stored), TN_INPUT_SELECT_POPUP.TcPOU (not stored), TN_INPUT_SELECT_TEXT.TcPOU (not stored), TN_RECEIVE.TcPOU (not stored), TN_SC_ADD_SHADOW.TcPOU (not stored), TN_SC_AREA_RESTORE.TcPOU (not stored), TN_SC_AREA_SAVE.TcPOU (not stored), TN_SC_BOX.TcPOU (not stored), TN_SC_FILL.TcPOU (not stored), TN_SC_LINE.TcPOU (not stored), TN_SC_READ_ATTR.TcPOU (not stored), TN_SC_READ_CHAR.TcPOU (not stored), TN_SC_SHADOW_ATTR.TcPOU (not stored), TN_SC_VIEWPORT.TcPOU (not stored), TN_SC_WRITE.TcPOU (not stored), TN_SC_WRITE_ATTR.TcPOU (not stored), TN_SC_WRITE_C.TcPOU (not stored), TN_SC_WRITE_CHAR.TcPOU (not stored), TN_SC_WRITE_EOS.TcPOU (not stored), TN_SC_XY2_ERROR.TcPOU (not stored), TN_SC_XY_ERROR.TcPOU (not stored), TN_SEND_ROWS.TcPOU (not stored)
//   oscat_network/POUs/WEATHER/ MOON_PHASE.TcPOU (not stored), WORLD_WEATHER.TcPOU (not stored), WORLD_WEATHER_DESC_GE.TcPOU (not stored), WORLD_WEATHER_ICON_OSCAT.TcPOU (not stored), YAHOO_WEATHER.TcPOU (not stored), YAHOO_WEATHER_DESC_GE.TcPOU (not stored), YAHOO_WEATHER_ICON_OSCAT.TcPOU (not stored)

// ---- oscat_basic/POUs/Engineering/signal processing/FILTER_MAV_DW.TcPOU
FUNCTION_BLOCK FILTER_MAV_DW
VAR_INPUT
	X : DWORD;
	N : UINT;
	RST : BOOL;
END_VAR
VAR_OUTPUT
	Y : DWORD;
END_VAR
VAR
	init : BOOL;
	buffer : ARRAY[0..31] OF DWORD;
	i : INT;
	sum : LWORD; 
END_VAR
VAR
	tmp: INT;
END_VAR

(*
version 1.3	23. feb. 2009
programmer 	hugo
tested by		oscat

FILTER_MAV_DW is a moving average filter with programmable length N for DWORD Data.
 
*)

(* limit N to size of buffer *)
N := MIN(N, 32);

(* startup initialisation *)
IF NOT init OR rst OR N = 0 THEN
	init := TRUE;
	tmp := UINT_TO_INT(N)-1;
	FOR i := 0 TO tmp DO
		buffer[i] := X;
	END_FOR;
	sum := Y * N;
	Y := X;
ELSE
	tmp := UINT_TO_INT(N);
	i := INC1(i, tmp);
	sum := sum + X - buffer[i];
	Y := LWORD_TO_DWORD(sum / N);
	buffer[i] := X;
END_IF;




(*
hm 13. oct. 2008	rev 1.0
	original version

hm	27. oct. 2008	rev 1.1
	added typecast to avoid warnings

hm	24. nov. 2008	rev 1.2
	added typecasts to avoid warnings
	avoid divide by 0 if N = 0

hm	23. feb. 2009	rev 1.3
	limit N to max array size

*)

END_FUNCTION_BLOCK
